% RSLogix 500 project Project 7.RSS, saved by version 8.30.00.16 %
PROJECT "UNTITLED"    % processor: Bul.1763 MicroLogix 1100 Series B %

PROGRAM FILES
  LAD 2   13 rungs

DATA FILES
  O0 OUTPUT  6 elements
  I1 INPUT  12 elements
  S2 STATUS  66 elements
  B3 BINARY  1 elements
  T4 TIMER  4 elements
  C5 COUNTER  2 elements
  R6 CONTROL  1 elements
  N7 INTEGER  9 elements
  F8 FLOAT  4 elements
  PD9 PID  1 elements

LADDER 2
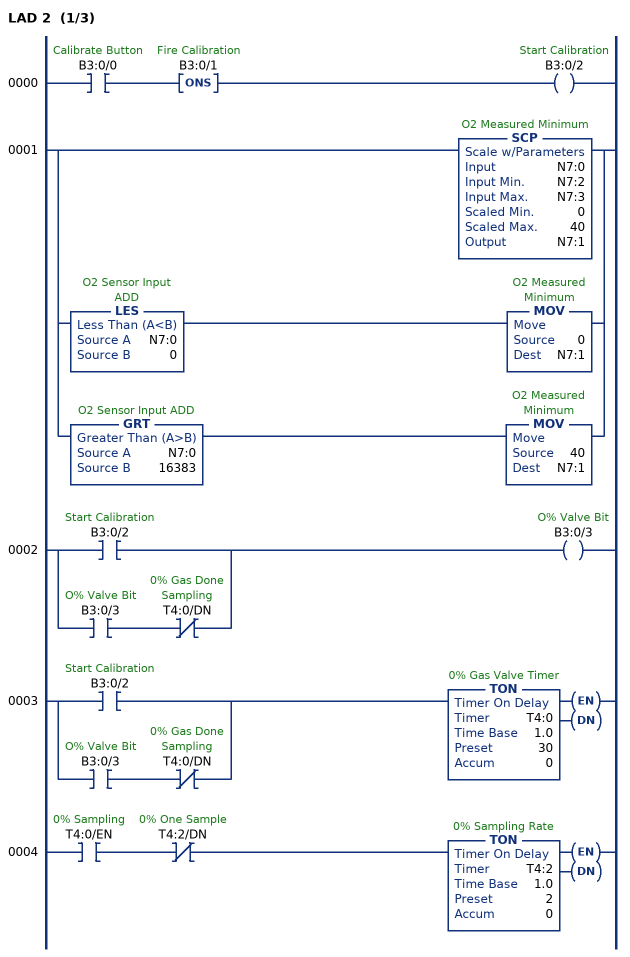
% Rung: 0 %
SOR XIC B3:0/0 ONS B3:0/1 OTE B3:0/2 EOR
%   B3:0/0  "Calibrate Button" %
%   B3:0/1  "Fire Calibration" %
%   B3:0/2  "Start Calibration" %
% Rung: 1 %
SOR BST SCP N7:0 N7:2 N7:3 0 40 N7:1 NXB LES N7:0 0 MOV 0 N7:1 NXB GRT N7:0 16383 MOV 40 N7:1 BND EOR
%   N7:0  ADD  "O2 Sensor Input" %
%   N7:2  "O2 Input Minimum" %
%   N7:3  "O2 Input Maximum" %
%   N7:1  "O2 Measured Minimum" %
% Rung: 2 %
SOR BST XIC B3:0/2 NXB XIC B3:0/3 XIO T4:0/DN BND OTE B3:0/3 EOR
%   B3:0/2  "Start Calibration" %
%   B3:0/3  "O% Valve Bit" %
%   T4:0/DN  "0% Gas Done Sampling" %
% Rung: 3 %
SOR BST XIC B3:0/2 NXB XIC B3:0/3 XIO T4:0/DN BND TON T4:0 1.0 30 0 EOR
%   B3:0/2  "Start Calibration" %
%   B3:0/3  "O% Valve Bit" %
%   T4:0/DN  "0% Gas Done Sampling" %
%   T4:0  "0% Gas Valve Timer" %
% Rung: 4 %
SOR XIC T4:0/EN XIO T4:2/DN TON T4:2 1.0 2 0 EOR
%   T4:0/EN  "0% Sampling" %
%   T4:2/DN  "0% One Sample" %
%   T4:2  "0% Sampling Rate" %

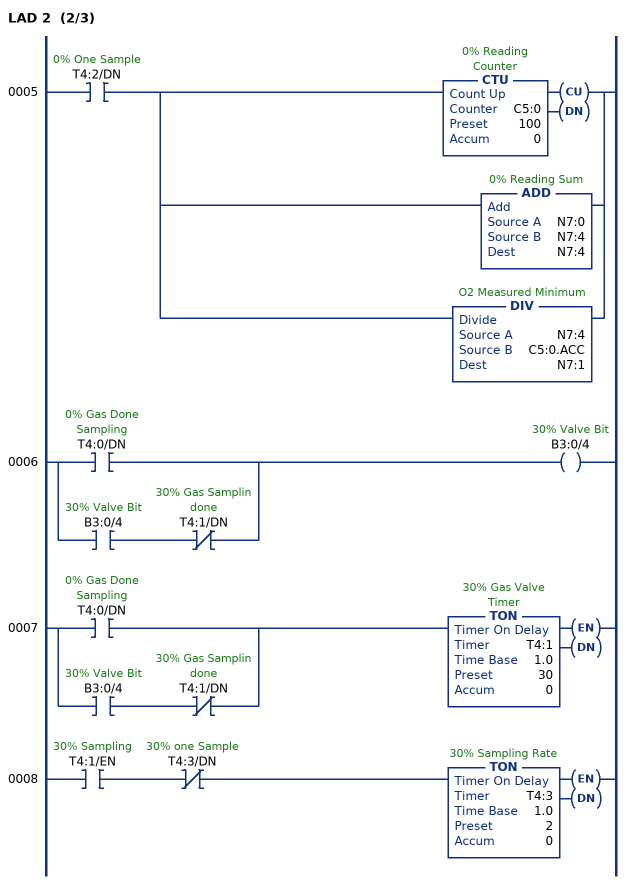
% Rung: 5 %
SOR XIC T4:2/DN BST CTU C5:0 100 0 NXB ADD N7:0 N7:4 N7:4 NXB DIV N7:4 C5:0.ACC N7:1 BND EOR
%   T4:2/DN  "0% One Sample" %
%   C5:0  "0% Reading Counter" %
%   N7:0  ADD  "O2 Sensor Input" %
%   N7:4  "0% Reading Sum" %
%   C5:0.ACC  "0% reading count" %
%   N7:1  "O2 Measured Minimum" %
% Rung: 6 %
SOR BST XIC T4:0/DN NXB XIC B3:0/4 XIO T4:1/DN BND OTE B3:0/4 EOR
%   T4:0/DN  "0% Gas Done Sampling" %
%   B3:0/4  "30% Valve Bit" %
%   T4:1/DN  "30% Gas Samplin done" %
% Rung: 7 %
SOR BST XIC T4:0/DN NXB XIC B3:0/4 XIO T4:1/DN BND TON T4:1 1.0 30 0 EOR
%   T4:0/DN  "0% Gas Done Sampling" %
%   B3:0/4  "30% Valve Bit" %
%   T4:1/DN  "30% Gas Samplin done" %
%   T4:1  "30% Gas Valve Timer" %
% Rung: 8 %
SOR XIC T4:1/EN XIO T4:3/DN TON T4:3 1.0 2 0 EOR
%   T4:1/EN  "30% Sampling" %
%   T4:3/DN  "30% one Sample" %
%   T4:3  "30% Sampling Rate" %

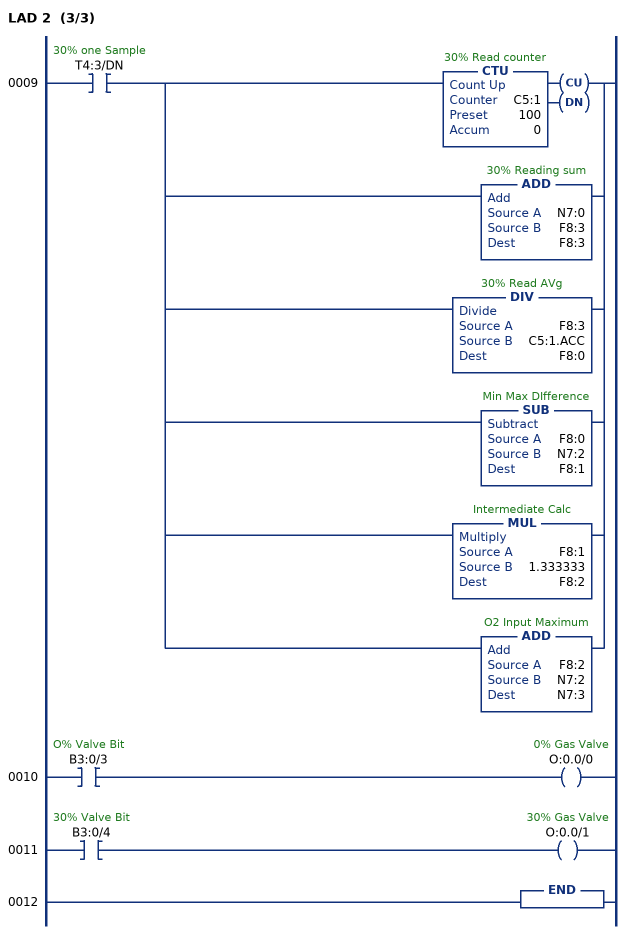
% Rung: 9 %
SOR XIC T4:3/DN BST CTU C5:1 100 0 NXB ADD N7:0 F8:3 F8:3 NXB DIV F8:3 C5:1.ACC F8:0 NXB SUB F8:0 N7:2 F8:1 NXB MUL F8:1 1.333333 F8:2 NXB ADD F8:2 N7:2 N7:3 BND EOR
%   T4:3/DN  "30% one Sample" %
%   C5:1  "30% Read counter" %
%   N7:0  ADD  "O2 Sensor Input" %
%   F8:3  "30% Reading sum" %
%   C5:1.ACC  "30% Reading Count" %
%   F8:0  "30% Read AVg" %
%   N7:2  "O2 Input Minimum" %
%   F8:1  "Min Max DIfference" %
%   F8:2  "Intermediate Calc" %
%   N7:3  "O2 Input Maximum" %
% Rung: 10 %
SOR XIC B3:0/3 OTE O:0.0/0 EOR
%   B3:0/3  "O% Valve Bit" %
%   O:0.0/0  "0% Gas Valve" %
% Rung: 11 %
SOR XIC B3:0/4 OTE O:0.0/1 EOR
%   B3:0/4  "30% Valve Bit" %
%   O:0.0/1  "30% Gas Valve" %
% Rung: 12 %
SOR END EOR

OTHER DOCUMENTED ADDRESSES
  B3:0/5  "Start Sampling"
  B3:0/6  "Start Averaging"
  B3:0/7  "Start averaging 30"
  N7:5  "30% read sum"
  N7:6  "30% Read Average"
  N7:7  "Max Min Diff"
  N7:8  "Intermediate Calc"
  N10:[C5:0.ACC]  "Sensor Read Storage"
  N11:[C5:0.ACC]  "30% Read Values"
  N11:[C5:1.ACC]  "30% Read value count"
  PD9:0  "PID FILE"
  T4:0/1  "30% Gas Valve Timer"
  T4:2/EN  "0% Sampling"

DATA TABLE (non-zero values as saved)
DATA T4
% .PRE .ACC %
% T4:0 % 30 0
% T4:1 % 30 0
% T4:2 % 2 0
% T4:3 % 2 0
DATA C5
% .PRE .ACC %
% C5:0 % 100 0
% C5:1 % 100 0
DATA N7
% N7:0 % 0 0 0 16383 0 0 0 0 0
